FUNCTION_BLOCK BfbOnePedCtrl
  (* Standard: 61499-2 *)
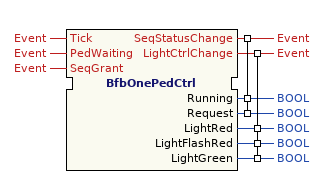
  EVENT_INPUT
    Tick;
    PedWaiting;
    SeqGrant;
  END_EVENT
  EVENT_OUTPUT
    SeqStatusChange WITH Running, Request;
    LightCtrlChange WITH LightRed, LightFlashRed, LightGreen;
  END_EVENT
  VAR_OUTPUT
    Running : BOOL := 0;
    Request : BOOL := 0;
    LightRed : BOOL := 0;
    LightFlashRed : BOOL := 0;
    LightGreen : BOOL := 0;
  END_VAR
  VAR
    d : UDINT := 0;
    greenTicks : UDINT := 10000000;
    flashTicks : UDINT := 10000000;
  END_VAR
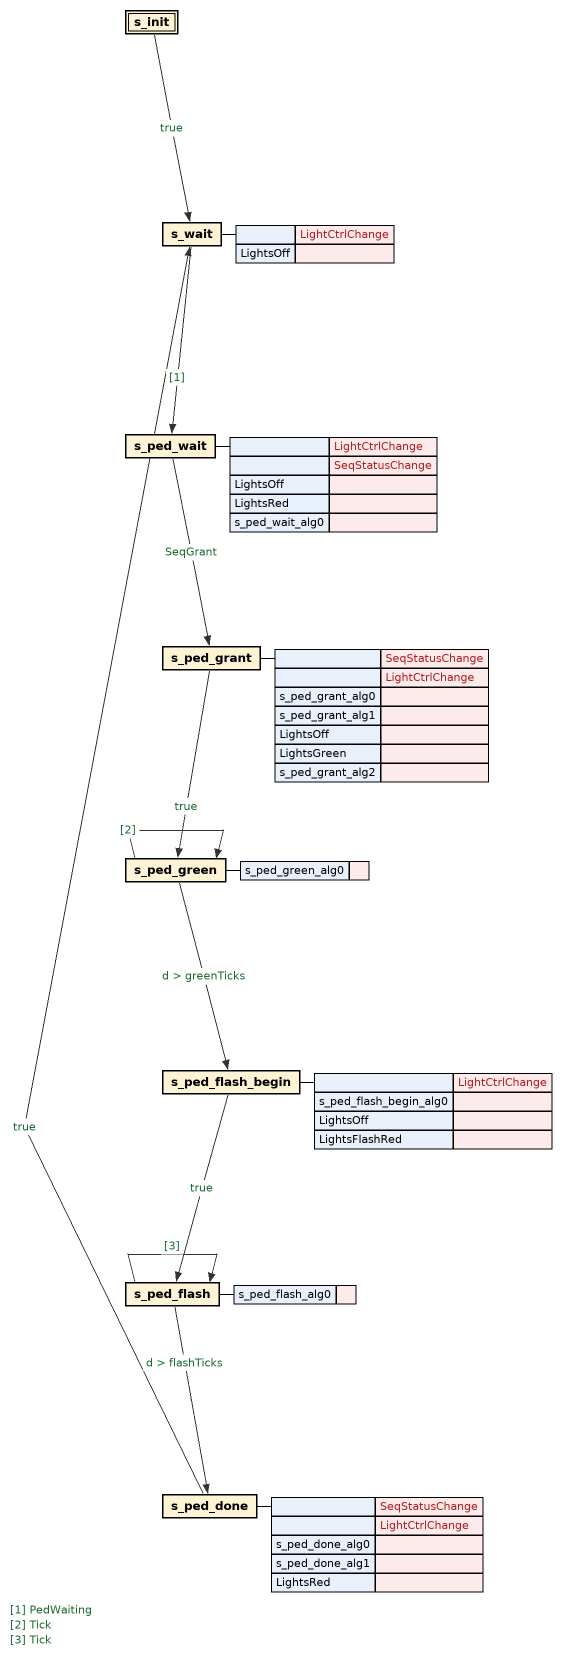
  EC_STATES
    s_init;
    s_wait : -> LightCtrlChange, LightsOff;
    s_ped_wait : -> LightCtrlChange, -> SeqStatusChange, LightsOff, LightsRed, s_ped_wait_alg0;
    s_ped_grant : -> SeqStatusChange, -> LightCtrlChange, s_ped_grant_alg0, s_ped_grant_alg1, LightsOff, LightsGreen, s_ped_grant_alg2;
    s_ped_green : s_ped_green_alg0;
    s_ped_flash_begin : -> LightCtrlChange, s_ped_flash_begin_alg0, LightsOff, LightsFlashRed;
    s_ped_flash : s_ped_flash_alg0;
    s_ped_done : -> SeqStatusChange, -> LightCtrlChange, s_ped_done_alg0, s_ped_done_alg1, LightsRed;
  END_STATES
  EC_TRANSITIONS
    s_init TO s_wait := true;
    s_wait TO s_ped_wait := PedWaiting;
    s_ped_wait TO s_ped_grant := SeqGrant;
    s_ped_grant TO s_ped_green := true;
    s_ped_green TO s_ped_flash_begin := d > greenTicks;
    s_ped_green TO s_ped_green := Tick;
    s_ped_flash_begin TO s_ped_flash := true;
    s_ped_flash TO s_ped_done := d > flashTicks;
    s_ped_flash TO s_ped_flash := Tick;
    s_ped_done TO s_wait := true;
  END_TRANSITIONS
  ALGORITHM s_ped_wait_alg0 IN ST:
Request := 1;
  END_ALGORITHM
  ALGORITHM s_ped_grant_alg0 IN ST:
Request := 0;
  END_ALGORITHM
  ALGORITHM s_ped_grant_alg1 IN ST:
Running := 1;
  END_ALGORITHM
  ALGORITHM s_ped_grant_alg2 IN ST:
d := 0;
  END_ALGORITHM
  ALGORITHM s_ped_green_alg0 IN ST:
d := d + 1
  END_ALGORITHM
  ALGORITHM s_ped_flash_begin_alg0 IN ST:
d := 0;
  END_ALGORITHM
  ALGORITHM s_ped_flash_alg0 IN ST:
d := d + 1;
  END_ALGORITHM
  ALGORITHM s_ped_done_alg0 IN ST:
Running := 0;
  END_ALGORITHM
  ALGORITHM s_ped_done_alg1 IN ST:
d := 0;
  END_ALGORITHM
  ALGORITHM LightsOff IN ST:
        LightRed := 0;
        LightFlashRed := 0;
        LightGreen := 0;
  END_ALGORITHM
  ALGORITHM LightsRed IN ST:
        LightRed := 1;
  END_ALGORITHM
  ALGORITHM LightsFlashRed IN ST:
        LightFlashRed := 1;
  END_ALGORITHM
  ALGORITHM LightsGreen IN ST:
        LightGreen := 1;
  END_ALGORITHM
END_FUNCTION_BLOCK
